TYPE "MaterialGateUDT"
VERSION : 0.1
   STRUCT
      CMD : Struct
         RequestPB : Bool;
         RequestPB_Auto : Bool;
      END_STRUCT;
      Status : Struct
         "Lock/Unlock Indicator" : Bool;
         "INT" : Int;
         Locked : Bool;
         Unlocked : Bool;
         Opened : Bool;
      END_STRUCT;
   END_STRUCT;

END_TYPE

